FUNCTION F_GetCycleTime : LREAL
VAR_INPUT
END_VAR
VAR
	fbTask:				GETCURTASKINDEX;
END_VAR

fbTask();
F_GetCycleTime:= UDINT_TO_LREAL(TwinCAT_SystemInfoVarList._TaskInfo[fbTask.index].CycleTime) / 10000000;

END_FUNCTION

(* stored: Version 1.1.0.1
   POU F_GetCycleTime: Id {249fe45c-5437-0e8d-0016-a00ccb17390e}, SpecialFunc None *)
